(* CoDeSys 2.3.9.62 project: DosCarritosLD v0.pro *)
(* Libraries: Standard.lib 2.6.14 10:37:46, IecSfc.lib 2.6.14 10:37:46 *)

(* Global variable list: Global_Variables *)
VAR_GLOBAL

      (*Entradas*)
      START:BOOL;
	A1:BOOL;
	B1:BOOL;
	A2:BOOL;
	B2:BOOL;
	M1:BOOL;
	M2:BOOL;

       (* Salidas *)
	MOTOR_IZ1:BOOL;
	MOTOR_DE1:BOOL;
       MOTOR_IZ2:BOOL;
	MOTOR_DE2:BOOL;

      (* Variables del simulador *)
	Vel:INT:=1;
	Vel2:INT:=1;
END_VAR

(* POU PLC_PRG, FBD *)
PROGRAM PLC_PRG
VAR

END_VAR
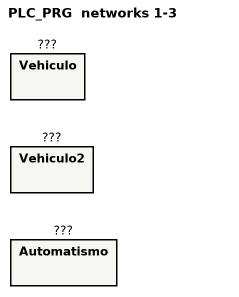
_FBD_ (* Function Block Diagram *)
NETWORK 1
	???:Vehiculo()
NETWORK 2
	???:Vehiculo2()
NETWORK 3
	???:Automatismo()
_END_FBD_
END_PROGRAM

(* POU Vehiculo, ST *)
PROGRAM Vehiculo
VAR
	PosX: INT;
END_VAR
A1:=FALSE;
B1:=FALSE;


IF MOTOR_DE1=TRUE THEN

     PosX:=PosX+Vel;

END_IF

IF MOTOR_IZ1=TRUE THEN

     PosX:=PosX-Vel;

END_IF


IF PosX<=0 THEN
   A1:=TRUE;
END_IF

IF PosX>=400 THEN
  B1:=TRUE;
END_IF
END_PROGRAM

(* POU Vehiculo2, ST *)
PROGRAM Vehiculo2
VAR
	PosX2: INT;
END_VAR
A2:=FALSE;
B2:=FALSE;


IF MOTOR_DE2=TRUE THEN

     PosX2:=PosX2+Vel2;

END_IF

IF MOTOR_IZ2=TRUE THEN

     PosX2:=PosX2-Vel2;

END_IF


IF PosX2<=0 THEN
   A2:=TRUE;
END_IF

IF PosX2>=400 THEN
  B2:=TRUE;
END_IF
END_PROGRAM

(* POU Automatismo, LD *)
PROGRAM Automatismo
VAR
	Vagoneta1: Vagoneta;		(*Increible se parece a su padre
			*)
	Vagoneta2: Vagoneta;
	VuelveYa: BOOL;
END_VAR
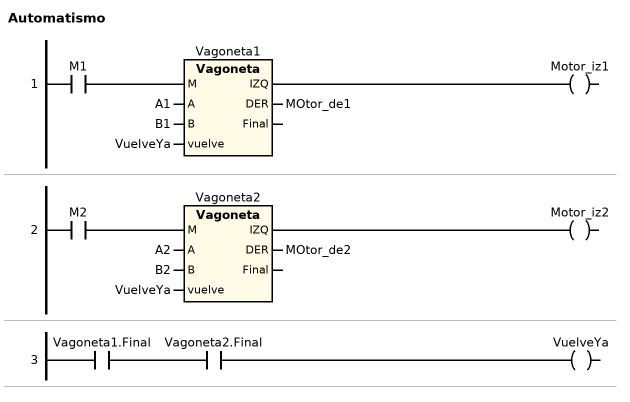
_LD_ (* Ladder Diagram *)
NETWORK 1
	[M1] - Vagoneta1:Vagoneta(M: *, A: A1, B: B1, vuelve: VuelveYa, DER => MOtor_de1) --- (Motor_iz1)
NETWORK 2
	[M2] - Vagoneta2:Vagoneta(M: *, A: A2, B: B2, vuelve: VuelveYa, DER => MOtor_de2) --- (Motor_iz2)
NETWORK 3
	[Vagoneta1.Final] - [Vagoneta2.Final] --- (VuelveYa)
_END_LD_
(* the same logic as Structured Text *)
(* Network 1 *)
Vagoneta1(M := M1, A := A1, B := B1, vuelve := VuelveYa);
MOtor_de1 := Vagoneta1.DER;
Motor_iz1 := Vagoneta1.IZQ;
(* Network 2 *)
Vagoneta2(M := M2, A := A2, B := B2, vuelve := VuelveYa);
MOtor_de2 := Vagoneta2.DER;
Motor_iz2 := Vagoneta2.IZQ;
(* Network 3 *)
VuelveYa := Vagoneta1.Final AND Vagoneta2.Final;
END_PROGRAM

(* POU Vagoneta, LD *)
FUNCTION_BLOCK Vagoneta
VAR_INPUT
	M:BOOL;
	A:BOOL;
	B:BOOL;
	vuelve:BOOL;

END_VAR
VAR_OUTPUT
	IZQ:BOOL;
	DER:BOOL;
	Final:BOOL;

END_VAR
VAR
END_VAR
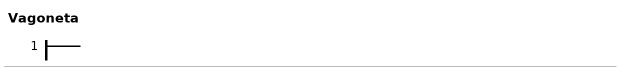
_LD_ (* Ladder Diagram *)
NETWORK 1
	*
_END_LD_
(* the same logic as Structured Text *)
(* Network 1 *)
END_FUNCTION_BLOCK

(* Visualisation Vehiculo
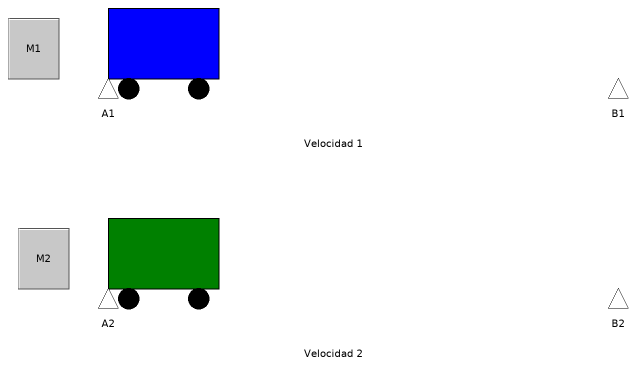
rectangle at (140,120)-(251,191): x offset Vehiculo.PosX
polygon at (130,190)-(150,210): alarm colour if .A1
polygon at (640,190)-(660,210): alarm colour if .B1
button at (40,130)-(91,191): text "M1"; taps M1
rectangle at (140,330)-(251,401): x offset Vehiculo2.PosX2
polygon at (130,400)-(150,420): alarm colour if .A2
polygon at (640,400)-(660,420): alarm colour if .B2
ellipse at (150,190)-(171,211): x offset Vehiculo.PosX
ellipse at (220,190)-(241,211): x offset Vehiculo.PosX
ellipse at (150,400)-(171,421): x offset Vehiculo2.PosX2
ellipse at (220,400)-(241,421): x offset Vehiculo2.PosX2
rectangle at (310,240)-(421,271): text "Velocidad 1"
rectangle at (310,450)-(421,481): text "Velocidad 2"
rectangle at (120,210)-(161,241): text "A1"
rectangle at (120,420)-(161,451): text "A2"
rectangle at (630,210)-(671,241): text "B1"
rectangle at (630,420)-(671,451): text "B2"
button at (50,340)-(101,401): text "M2"; taps M2
2 elements of other kinds (tables, trends, ...) not read
*)
